PROGRAM MAIN
VAR
	Count : INT;
END_VAR

Count := 0;

END_PROGRAM

(* stored: Version 1.1.0.1, ProductVersion 3.1.4024.4
   POU MAIN: Id {583f6538-72a5-4bdd-a773-e6c25fe897e0}, SpecialFunc None *)
